FUNCTION_BLOCK FB_ExtruderControl
VAR_INPUT
	bHeatersEnabled	: BOOL;						// Heizelemente aktiviert
END_VAR
VAR_OUTPUT
	// Statusinformationen
	bReady 			: BOOL;						// Betriebsbereit auf Temperatur
	bExtruding 		: BOOL;						// Motor läuft
	bHeatingActiv 	: BOOL;						// Heizelemente
	bError        	: BOOL;						// Fehler
    nErrorID      	: UDINT;
    sErrorMsg 		: STRING(80);
END_VAR
VAR
	// Zustandsmaschine
	eState			: E_StateExtruder := E_StateExtruder.OFF;	//State
END_VAR
VAR_IN_OUT
	// Steuersignale
	bStartHeater 	: BOOL;						// Heizelemente aktivieren
	bStopHeater		: BOOL;						// Abschalten und Abkühlen
	bStart 			: BOOL;						// Start-Befehl Extrusion
	bStop 			: BOOL;						// Stop-Befehl Extrusion
	bErrorReset 	: BOOL;						// Reset-Befehl für Fehler
END_VAR

(*
	0   - Ausgeschaltet (OFF)
	10  - Initialisierung (INIT)
	100 - Warte auf Befehl (IDLE)
	200 - Aufheizen (HEATING)
	300 - Betriebsbereit (READY)
	310 - Motor aktiviert / Drucken (PRINTING)
	400 - Herunterfahren (SHUTDOWN)
*)

// =============================================================================
// Extrusionsrate berechnen
// =============================================================================
FC_ExtrusionCalculations();

// =============================================================================
// Funktionsabhängigkeiten (Heizen vor Extrusion und Stop dominant)
// =============================================================================
IF bStop THEN
	bStart := FALSE;
ELSIF bStart THEN
	bStartHeater := TRUE;
END_IF

IF bStopHeater OR NOT bHeatersEnabled THEN
	bStart := FALSE;
	bStop := TRUE;
	bStartHeater := FALSE;
END_IF

// =============================================================================
// Fehlerbahandlung
// =============================================================================
IF bErrorReset AND bError THEN
	GVL_Extruder.HeaterTop.bErrorReset := TRUE;
	GVL_Extruder.HeaterMiddle.bErrorReset := TRUE;
	GVL_Extruder.HeaterNozzle.bErrorReset := TRUE;
	GVL_Extruder.ExtruderMotor.bErrorReset := TRUE;
	bErrorReset := FALSE;
	bError := FALSE;
END_IF;

bError := bError
	OR GVL_Extruder.HeaterTop.bError 
	OR GVL_Extruder.HeaterMiddle.bError
	OR GVL_Extruder.HeaterNozzle.bError
	OR GVL_Extruder.ExtruderMotor.bError;
	
IF bError THEN
	IF GVL_Extruder.HeaterTop.bError 		THEN nErrorID := GVL_Extruder.HeaterTop.nErrorID + 10; END_IF
	IF GVL_Extruder.HeaterMiddle.bError 	THEN nErrorID := GVL_Extruder.HeaterMiddle.nErrorID + 20; END_IF
	IF GVL_Extruder.HeaterNozzle.bError 	THEN nErrorID := GVL_Extruder.HeaterNozzle.nErrorID + 30; END_IF
	IF GVL_Extruder.ExtruderMotor.bError 	THEN nErrorID := GVL_Extruder.ExtruderMotor.nErrorID; END_IF
	IF GVL_Extruder.HeaterTop.bError 		THEN sErrorMsg := GVL_Extruder.HeaterTop.sErrorMsg; END_IF
	IF GVL_Extruder.HeaterMiddle.bError 	THEN sErrorMsg := GVL_Extruder.HeaterMiddle.sErrorMsg; END_IF
	IF GVL_Extruder.HeaterNozzle.bError 	THEN sErrorMsg := GVL_Extruder.HeaterNozzle.sErrorMsg; END_IF
	IF GVL_Extruder.ExtruderMotor.bError 	THEN sErrorMsg := GVL_Extruder.ExtruderMotor.sErrorMsg; END_IF
END_IF

IF bError AND NOT (eState = E_StateExtruder.IDLE OR eState = E_StateExtruder.OFF) THEN
	eState := E_StateExtruder.SHUTDOWN;
END_IF

// =============================================================================
// Status
// =============================================================================
bExtruding := GVL_Extruder.ExtruderMotor.bRunning;

// =============================================================================
// Zustandsmaschine
// =============================================================================
CASE eState OF
	// =============================================================================
	E_StateExtruder.OFF : // Ausgeschaltet
	// =============================================================================
		// Alles aus
		GVL_Extruder.HeaterTop.bEnabled := FALSE;
		GVL_Extruder.HeaterMiddle.bEnabled := FALSE;
		GVL_Extruder.HeaterNozzle.bEnabled := FALSE;
		GVL_Extruder.ExtruderMotor.bEnable := FALSE;
	
		// Status
		bReady := FALSE;
		bHeatingActiv := FALSE;
		
		IF NOT bError THEN
			eState := E_StateExtruder.INIT;
		END_IF;
		
	// =============================================================================
	E_StateExtruder.INIT: // Initialisierung
	// =============================================================================
		eState := E_StateExtruder.IDLE;
	
	// =============================================================================
	E_StateExtruder.IDLE : // Idle
	// =============================================================================
		// Alles aus
		GVL_Extruder.HeaterTop.bEnabled := FALSE;
		GVL_Extruder.HeaterMiddle.bEnabled := FALSE;
		GVL_Extruder.HeaterNozzle.bEnabled := FALSE;
		GVL_Extruder.ExtruderMotor.bEnable := FALSE;
	
		// Status
		bReady := FALSE;
		bHeatingActiv := FALSE;
		
		IF bStartHeater 
		AND (GVL_ParameterExtruder.aMaterialSettings[GVL_ParameterExtruder.nMaterial].fTempTop 		<> 0.0 
			OR GVL_ParameterExtruder.aMaterialSettings[GVL_ParameterExtruder.nMaterial].fTempMiddle <> 0.0 
			OR GVL_ParameterExtruder.aMaterialSettings[GVL_ParameterExtruder.nMaterial].fTempNozzle <> 0.0) 
		AND NOT bStopHeater AND bHeatersEnabled THEN
			eState := E_StateExtruder.HEATING;
		END_IF;
		
	// =============================================================================
	E_StateExtruder.HEATING : // Aufheizen
	// =============================================================================
		// Starte Heizelemente
		GVL_Extruder.HeaterTop.bEnabled := TRUE;
		GVL_Extruder.HeaterMiddle.bEnabled := TRUE;
		GVL_Extruder.HeaterNozzle.bEnabled := TRUE;
		GVL_Extruder.ExtruderMotor.bEnable := FALSE;
		
		//Status
		bReady := FALSE;
		bHeatingActiv := TRUE;
		
		// Prüfe, ob alle Temperaturen erreicht
		IF bStopHeater OR NOT bHeatersEnabled THEN
			eState := E_StateExtruder.SHUTDOWN;
		ELSIF (GVL_Extruder.HeaterTop.bAtTemp OR GVL_ParameterExtruder.aMaterialSettings[GVL_ParameterExtruder.nMaterial].fTempTop = 0.0)
		AND (GVL_Extruder.HeaterMiddle.bAtTemp OR GVL_ParameterExtruder.aMaterialSettings[GVL_ParameterExtruder.nMaterial].fTempMiddle = 0.0)
		AND (GVL_Extruder.HeaterNozzle.bAtTemp OR GVL_ParameterExtruder.aMaterialSettings[GVL_ParameterExtruder.nMaterial].fTempNozzle = 0.0) THEN
			eState := E_StateExtruder.READY;
		END_IF
	
	// =============================================================================
	E_StateExtruder.READY: // Betriebsbereit, Heizelemente aktiv
	// =============================================================================
		//Status
		bReady := TRUE;
		bHeatingActiv := TRUE;
		
		// Heizelemente aktiv
		GVL_Extruder.HeaterTop.bEnabled := TRUE;
		GVL_Extruder.HeaterMiddle.bEnabled := TRUE;
		GVL_Extruder.HeaterNozzle.bEnabled := TRUE;
		GVL_Extruder.ExtruderMotor.bEnable := FALSE;

		IF bStopHeater OR NOT bHeatersEnabled THEN
			eState := E_StateExtruder.SHUTDOWN;
		ELSIF bStart THEN
			eState := E_StateExtruder.PRINTING;
		END_IF;
	
	// =============================================================================
	E_StateExtruder.PRINTING : // Motor aktiviert / Extrusion
	// =============================================================================
		// Halte Heizungen aktiv
		GVL_Extruder.HeaterTop.bEnabled := TRUE;
		GVL_Extruder.HeaterMiddle.bEnabled := TRUE;
		GVL_Extruder.HeaterNozzle.bEnabled := TRUE;
		
		// Motor starten
		GVL_Extruder.ExtruderMotor.bEnable := TRUE;
		
		//Status
		bReady := TRUE;
		bHeatingActiv := TRUE;
		
		IF bStopHeater OR NOT bHeatersEnabled THEN
			eState := E_StateExtruder.SHUTDOWN;		
		ELSIF bStop THEN
			GVL_Extruder.ExtruderMotor.bEnable := FALSE;
			eState := E_StateExtruder.READY;
		END_IF;
	
	// =============================================================================
	E_StateExtruder.SHUTDOWN : // Herunterfahren
	// =============================================================================
		// Schalte alles ab
		GVL_Extruder.HeaterTop.bEnabled := FALSE;
		GVL_Extruder.HeaterMiddle.bEnabled := FALSE;
		GVL_Extruder.HeaterNozzle.bEnabled := FALSE;

		GVL_Extruder.ExtruderMotor.bEnable := FALSE;
		
		// Status
		bReady := FALSE;
		bHeatingActiv := FALSE;
		
		// Cooldown Bedingung (alles unter 35°C)
		IF GVL_Extruder.HeaterTop.fActualTemp < 35
		AND GVL_Extruder.HeaterMiddle.fActualTemp < 35
		AND GVL_Extruder.HeaterNozzle.fActualTemp < 35 THEN
			eState := E_StateExtruder.IDLE;
		ELSIF (GVL_ParameterExtruder.aMaterialSettings[GVL_ParameterExtruder.nMaterial].fTempTop 	<> 0.0 
		OR GVL_ParameterExtruder.aMaterialSettings[GVL_ParameterExtruder.nMaterial].fTempMiddle <> 0.0 
		OR GVL_ParameterExtruder.aMaterialSettings[GVL_ParameterExtruder.nMaterial].fTempNozzle <> 0.0) 
		AND NOT bError AND bStartHeater AND NOT bStopHeater AND bHeatersEnabled THEN
			eState := E_StateExtruder.HEATING;
		END_IF;
END_CASE;

END_FUNCTION_BLOCK

(* stored: Version 1.1.0.1
   POU FB_ExtruderControl: Id {83cefcd4-2bc0-4963-a2a0-3b0dcab13e7f}, SpecialFunc None *)
